// Mitsubishi GX Works2 project: TEx03   PLC: Q02/Q02H

PROGRAM MAIN
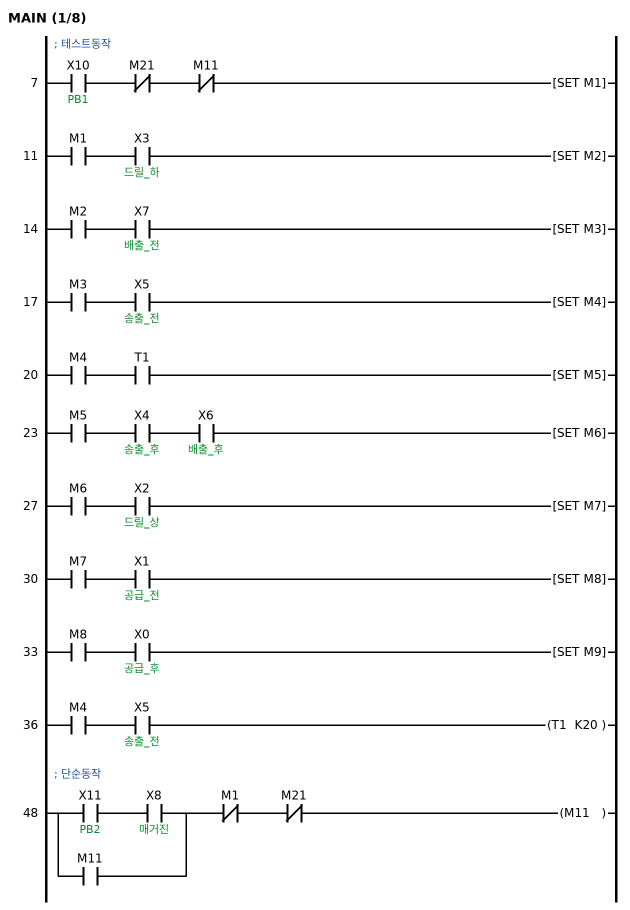
; 테스트동작
7     LD      X10  ; PB1
      ANI     M21
      ANI     M11
      SET     M1
11    LD      M1
      AND     X3  ; 드릴_하
      SET     M2
14    LD      M2
      AND     X7  ; 배출_전
      SET     M3
17    LD      M3
      AND     X5  ; 송출_전
      SET     M4
20    LD      M4
      AND     T1
      SET     M5
23    LD      M5
      AND     X4  ; 송출_후
      AND     X6  ; 배출_후
      SET     M6
27    LD      M6
      AND     X2  ; 드릴_상
      SET     M7
30    LD      M7
      AND     X1  ; 공급_전
      SET     M8
33    LD      M8
      AND     X0  ; 공급_후
      SET     M9
36    LD      M4
      AND     X5  ; 송출_전
      OUT     T1 K20
; 단순동작
48    LD      X11  ; PB2
      AND     X8  ; 매거진
      OR      M11
      ANI     M1
      ANI     M21
      OUT     M11
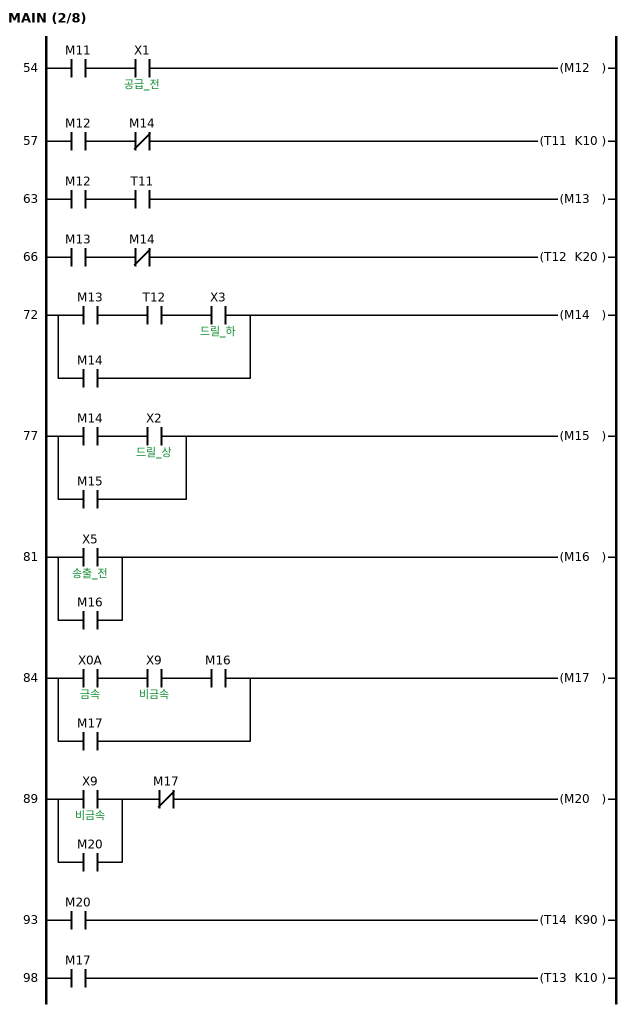
54    LD      M11
      AND     X1  ; 공급_전
      OUT     M12
57    LD      M12
      ANI     M14
      OUT     T11 K10
63    LD      M12
      AND     T11
      OUT     M13
66    LD      M13
      ANI     M14
      OUT     T12 K20
72    LD      M13
      AND     T12
      AND     X3  ; 드릴_하
      OR      M14
      OUT     M14
77    LD      M14
      AND     X2  ; 드릴_상
      OR      M15
      OUT     M15
81    LD      X5  ; 송출_전
      OR      M16
      OUT     M16
84    LD      X0A  ; 금속
      AND     X9  ; 비금속
      AND     M16
      OR      M17
      OUT     M17
89    LD      X9  ; 비금속
      OR      M20
      ANI     M17
      OUT     M20
93    LD      M20
      OUT     T14 K90
98    LD      M17
      OUT     T13 K10
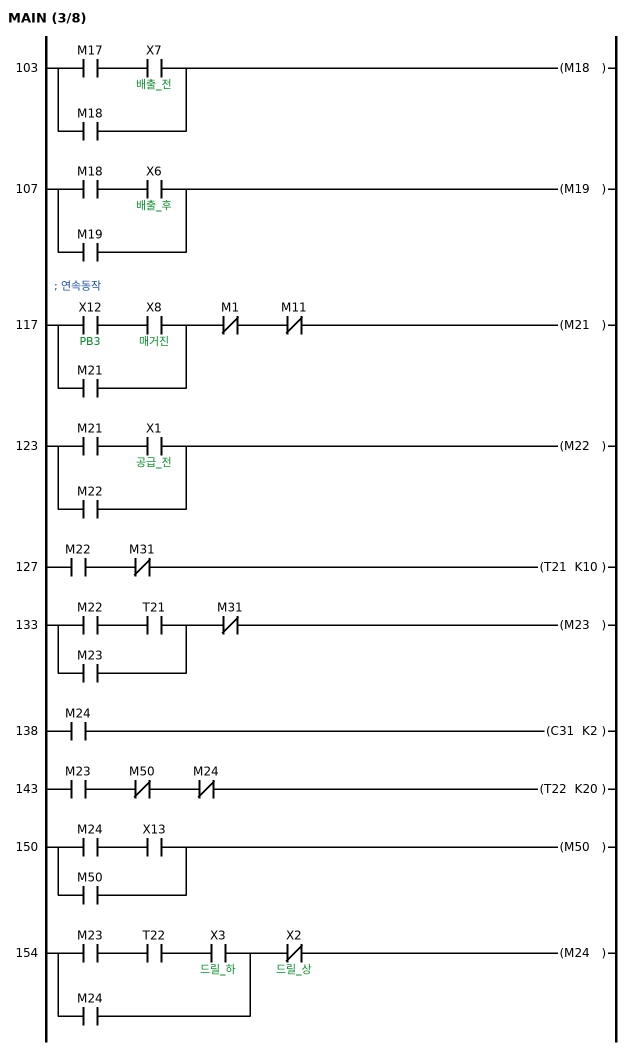
103   LD      M17
      AND     X7  ; 배출_전
      OR      M18
      OUT     M18
107   LD      M18
      AND     X6  ; 배출_후
      OR      M19
      OUT     M19
; 연속동작
117   LD      X12  ; PB3
      AND     X8  ; 매거진
      OR      M21
      ANI     M1
      ANI     M11
      OUT     M21
123   LD      M21
      AND     X1  ; 공급_전
      OR      M22
      OUT     M22
127   LD      M22
      ANI     M31
      OUT     T21 K10
133   LD      M22
      AND     T21
      OR      M23
      ANI     M31
      OUT     M23
138   LD      M24
      OUT     C31 K2
143   LD      M23
      ANI     M50
      ANI     M24
      OUT     T22 K20
150   LD      M24
      AND     X13
      OR      M50
      OUT     M50
154   LD      M23
      AND     T22
      AND     X3  ; 드릴_하
      OR      M24
      ANI     X2  ; 드릴_상
      OUT     M24
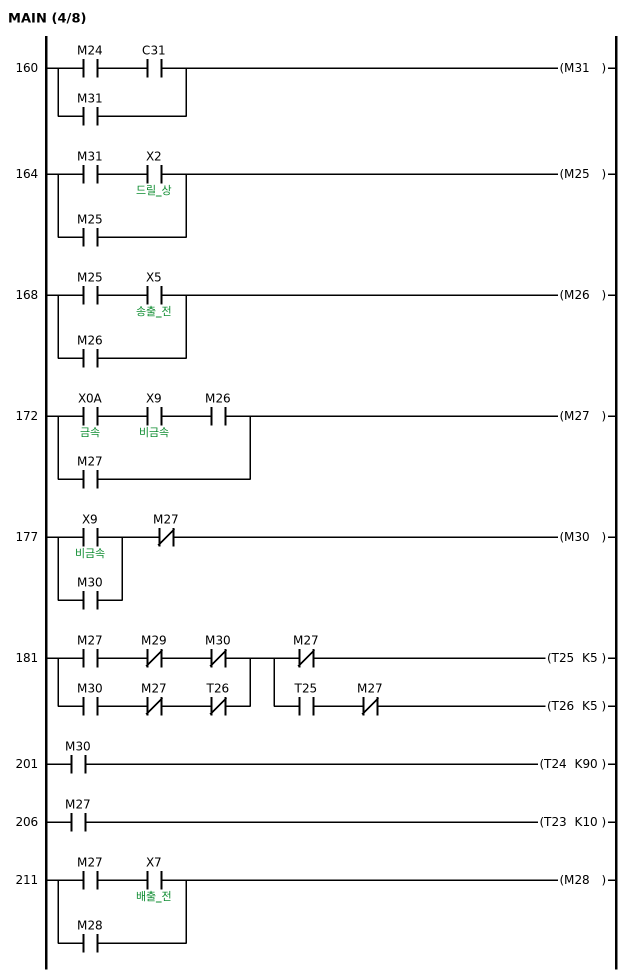
160   LD      M24
      AND     C31
      OR      M31
      OUT     M31
164   LD      M31
      AND     X2  ; 드릴_상
      OR      M25
      OUT     M25
168   LD      M25
      AND     X5  ; 송출_전
      OR      M26
      OUT     M26
172   LD      X0A  ; 금속
      AND     X9  ; 비금속
      AND     M26
      OR      M27
      OUT     M27
177   LD      X9  ; 비금속
      OR      M30
      ANI     M27
      OUT     M30
181   LD      M27
      ANI     M29
      ANI     M30
      LD      M30
      ANI     M27
      ANI     T26
      ORB
      MPS
      ANI     M27
      OUT     T25 K5
      MPP
      AND     T25
      ANI     M27
      OUT     T26 K5
201   LD      M30
      OUT     T24 K90
206   LD      M27
      OUT     T23 K10
211   LD      M27
      AND     X7  ; 배출_전
      OR      M28
      OUT     M28
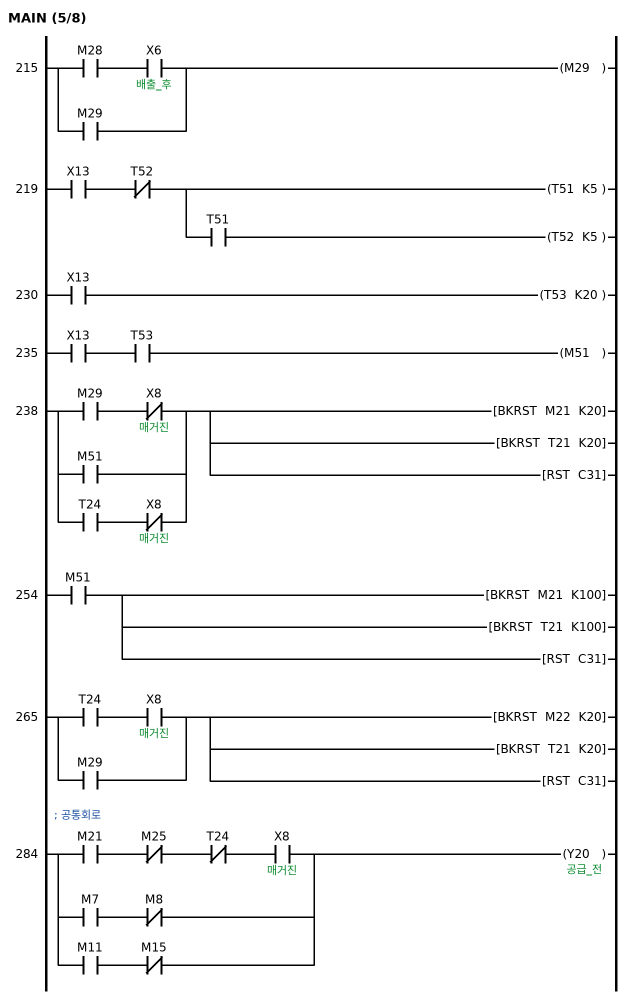
215   LD      M28
      AND     X6  ; 배출_후
      OR      M29
      OUT     M29
219   LD      X13
      ANI     T52
      OUT     T51 K5
      AND     T51
      OUT     T52 K5
230   LD      X13
      OUT     T53 K20
235   LD      X13
      AND     T53
      OUT     M51
238   LD      M29
      ANI     X8  ; 매거진
      OR      M51
      LD      T24
      ANI     X8  ; 매거진
      ORB
      BKRST   M21 K20
      BKRST   T21 K20
      RST     C31
254   LD      M51
      BKRST   M21 K100
      BKRST   T21 K100
      RST     C31
265   LD      T24
      AND     X8  ; 매거진
      OR      M29
      BKRST   M22 K20
      BKRST   T21 K20
      RST     C31
; 공통회로
284   LD      M21
      ANI     M25
      ANI     T24
      AND     X8  ; 매거진
      LD      M7
      ANI     M8
      ORB
      LD      M11
      ANI     M15
      ORB
      OUT     Y20  ; 공급_전
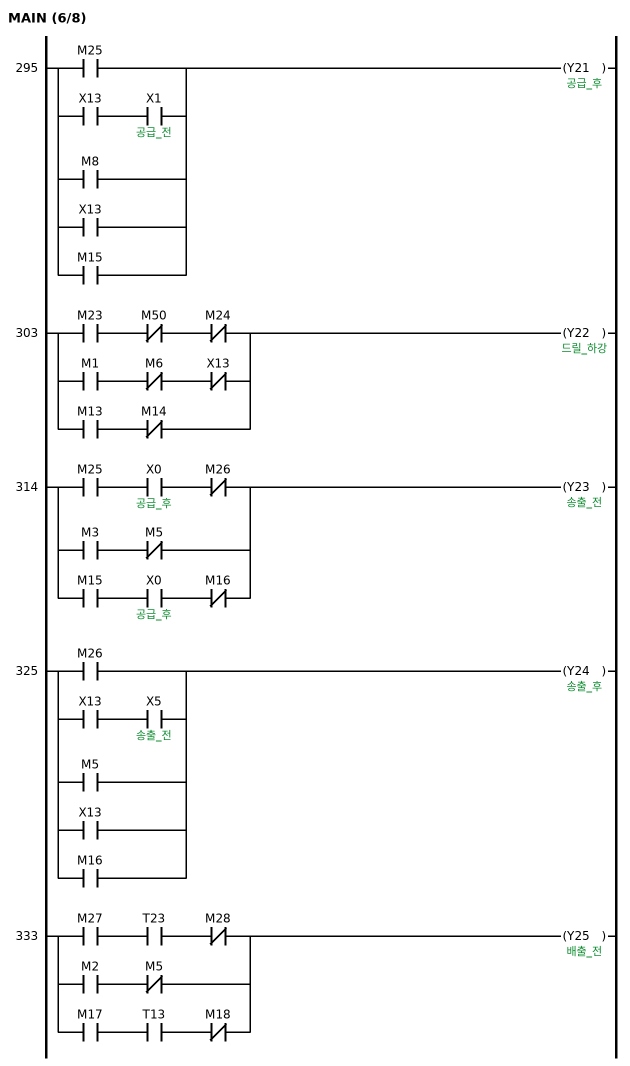
295   LD      M25
      LD      X13
      AND     X1  ; 공급_전
      ORB
      OR      M8
      OR      X13
      OR      M15
      OUT     Y21  ; 공급_후
303   LD      M23
      ANI     M50
      ANI     M24
      LD      M1
      ANI     M6
      ANI     X13
      ORB
      LD      M13
      ANI     M14
      ORB
      OUT     Y22  ; 드릴_하강
314   LD      M25
      AND     X0  ; 공급_후
      ANI     M26
      LD      M3
      ANI     M5
      ORB
      LD      M15
      AND     X0  ; 공급_후
      ANI     M16
      ORB
      OUT     Y23  ; 송출_전
325   LD      M26
      LD      X13
      AND     X5  ; 송출_전
      ORB
      OR      M5
      OR      X13
      OR      M16
      OUT     Y24  ; 송출_후
333   LD      M27
      AND     T23
      ANI     M28
      LD      M2
      ANI     M5
      ORB
      LD      M17
      AND     T13
      ANI     M18
      ORB
      OUT     Y25  ; 배출_전
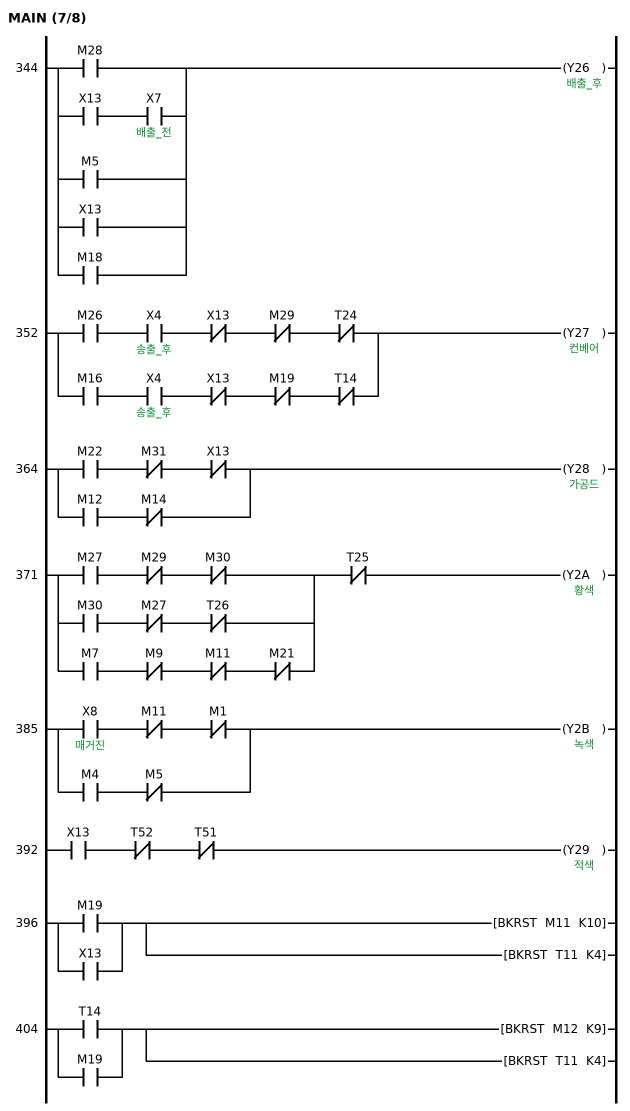
344   LD      M28
      LD      X13
      AND     X7  ; 배출_전
      ORB
      OR      M5
      OR      X13
      OR      M18
      OUT     Y26  ; 배출_후
352   LD      M26
      AND     X4  ; 송출_후
      ANI     X13
      ANI     M29
      ANI     T24
      LD      M16
      AND     X4  ; 송출_후
      ANI     X13
      ANI     M19
      ANI     T14
      ORB
      OUT     Y27  ; 컨베어
364   LD      M22
      ANI     M31
      ANI     X13
      LD      M12
      ANI     M14
      ORB
      OUT     Y28  ; 가공드
371   LD      M27
      ANI     M29
      ANI     M30
      LD      M30
      ANI     M27
      ANI     T26
      ORB
      LD      M7
      ANI     M9
      ANI     M11
      ANI     M21
      ORB
      ANI     T25
      OUT     Y2A  ; 황색
385   LD      X8  ; 매거진
      ANI     M11
      ANI     M1
      LD      M4
      ANI     M5
      ORB
      OUT     Y2B  ; 녹색
392   LD      X13
      ANI     T52
      ANI     T51
      OUT     Y29  ; 적색
396   LD      M19
      OR      X13
      BKRST   M11 K10
      BKRST   T11 K4
404   LD      T14
      OR      M19
      BKRST   M12 K9
      BKRST   T11 K4
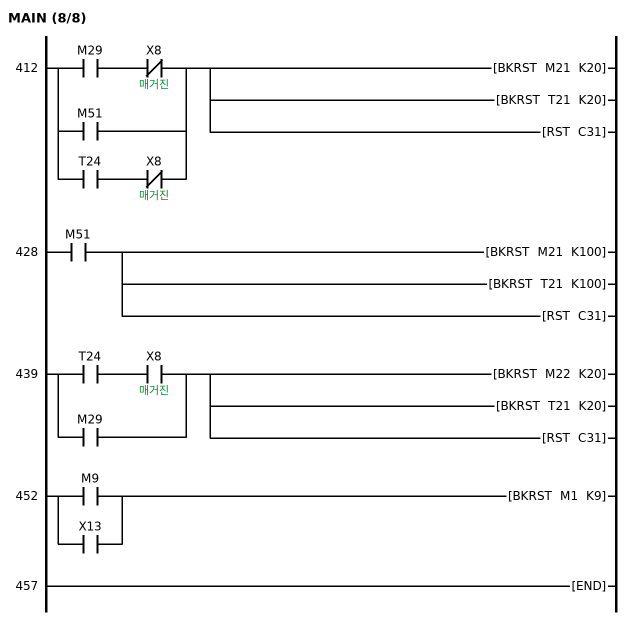
412   LD      M29
      ANI     X8  ; 매거진
      OR      M51
      LD      T24
      ANI     X8  ; 매거진
      ORB
      BKRST   M21 K20
      BKRST   T21 K20
      RST     C31
428   LD      M51
      BKRST   M21 K100
      BKRST   T21 K100
      RST     C31
439   LD      T24
      AND     X8  ; 매거진
      OR      M29
      BKRST   M22 K20
      BKRST   T21 K20
      RST     C31
452   LD      M9
      OR      X13
      BKRST   M1 K9
457   END
END_PROGRAM
